PROGRAM MAIN
VAR
END_VAR

END_PROGRAM

(* stored: Version 1.1.0.1
   POU MAIN: Id {eb951b9b-e79b-4e38-8d9d-01b9420706c0} *)
